// Block: DEBUG_MES_Receive_Msg_Topic1XX

DATA_BLOCK DEBUG_MES_Receive_Msg_Topic1XX
VERSION : 0.1
   NON_RETAIN
   VAR
      DEBUG : Struct
         Enable : Bool;
         AckChangeStep : Bool;
         ActualStep : Int;
      END_STRUCT;
      ACK_MSG_enable : Bool;
      MSG_100 : Struct
         ABILITA_FC : Bool;
         EXE_MSG_S060x40x125 : Bool;
         EXE_MSG_S120x45x125 : Bool;
         EXE_MSG_C060x40x125_L1000 : Bool;
         EXE_MSG_C060x40x125_L2000 : Bool;
         EXE_MSG_C060x40x125_L3000 : Bool;
         EXE_MSG_C140x45x125_L3000 : Bool;
         EXE_MSG_C120x45x125_L2700 : Bool;
         Msg_ID : DInt;
         MSG : MES_Msg;
      END_STRUCT;
      MSG_130 : Struct
         ABILITA_FC : Bool;
         EXE_MSG : Bool;
         IDP : String;
         MSG : MES_Msg;
      END_STRUCT;
      MSG_140 : Struct
         ABILITA_FC : Bool;
         EXE_MSG : Bool;
         IDP : String;
         MSG : MES_Msg;
      END_STRUCT;
      MSG_142 : Struct
         ABILITA_FC : Bool;
         EXE_MSG : Bool;
         MSG : MES_Msg;
      END_STRUCT;
      FUN : Struct
         ABILITA_FC : Bool;
         RETVAL : DInt;
         EXE_Copy_From_RECEIVE_TOPIC_100 : Bool;
         Prod_Item : Prod_Item;
         CHECK_ITEM_VALID : Struct
            EXE : Bool;
         END_STRUCT;
         GET_BY_IDP_MES : Struct
            EXE : Bool;
            MES_IDP : String;
            RETVAL : DInt;
            item_Prod : Prod_Item;
            Index : Int;
         END_STRUCT;
      END_STRUCT;
   END_VAR

BEGIN
   // No initialization required
END_DATA_BLOCK
